TYPE "nodeLinkSourceToDest"
TITLE = {"version":"v1.1","author":"cyanezf","family":"core/node","status":"deprecated","deprecatedBy": "nodeLinkSourceToDest-v1.2","dependencies":[]}

//(*--
//# Documentation
//## Log
//| version | date | author | description |
//|:-------:|:----:|:------:|:------------|
//| v1.1 | 2023-10-20 | cyanezf | `shortCycle` added |
//| v1.0 | 2023-10-19 | cyanezf | First version |
//
//## Description
//Node link - source to destination
//--*)

   STRUCT
      transferring : Bool;   // 1=Transferring object
      shortCycle : Bool;   // 1=Short cycle
   END_STRUCT;

END_TYPE

